PROGRAM Transformer
VAR_INPUT
	// reset signal for the error condition
	reset_error:		BOOL := FALSE;
	// signal to start the transformer
	softstart_trafo:	BOOL;
END_VAR
VAR_OUTPUT
	// indicates the phases for the hydraulics
	phase_available:	BOOL;
	// trafo failed to start after timeout
	power_failure:		BOOL;
	// restart was inhibited
	restart_inhibited:	BOOL;
END_VAR
VAR
	// watchdog for trafo softstarter
	power_watchdog: 	TON;
	// timer to measure the startup time
	power_timer:		FB_timer;
	// timeout for the startup
	startup_timeout:	TIME := T#5S;
	// error state
	power_error_state:	SR;
	// restart inhibitor
	restart_inhibit:	TOF;
	PowerEvent:			FB_EventLog;
	PowerLog:			FB_EventLog;
END_VAR

power_timer(bStart := GVL_Main.softstart_trafo, bStop := power_OK);
power_watchdog(IN := GVL_Main.softstart_trafo AND NOT power_OK,
				PT := startup_timeout,
				Q => power_failure);
power_error_state(SET1 := power_failure, RESET := reset_error);
restart_inhibit(IN := GVL_MAIN.trafo_bypassed, PT := T#5S);

restart_inhibited := NOT GVL_MAIN.trafo_bypassed AND restart_inhibit.Q;
IF restart_inhibited THEN
	softstart_trafo := FALSE;
END_IF
GVL_Main.softstart_trafo := softstart_trafo AND NOT error;

phase_available := TRUE; (*GVL_Main.L1L2_voltage > 360.0 AND
					GVL_Main.L2L3_voltage > 360.0 AND
					GVL_Main.L3L1_voltage > 360.0; *)

PowerEvent(	
	Trigger := 		power_failure, 
	Level := 		ADSLOG_MSGTYPE_ERROR,
	FormatString :=	'%s',
	OnMessage := 	'Servo power FAILURE!',
	OffMEssage := 	'Servo power OK');
PowerLog(	
	Trigger := 		power_OK, 
	Level := 		ADSLOG_MSGTYPE_HINT,
	FormatString :=	'%s',
	OnMessage := 	'Mains power is ON',
	OffMEssage := 	'Mains power is OFF');

PROPERTY error : BOOL
GET
error := power_error_state.Q1;
END_GET
END_PROPERTY

PROPERTY power_ok : BOOL
// indicates the power state for the AX5000
GET
power_ok := GVL_main.trafo_bypassed;
END_GET
END_PROPERTY

METHOD reset : BOOL
VAR_INPUT
END_VAR
IF error THEN
	reset_error := TRUE;
ELSE
	reset_error := FALSE;
END_IF
END_METHOD

METHOD start : BOOL
VAR_INPUT
END_VAR
softstart_trafo := TRUE;
END_METHOD

PROPERTY startup_time : TIME
GET
startup_time := power_timer.tDifference;
END_GET
SET
startup_timeout := startup_time;
END_SET
END_PROPERTY

METHOD stop : BOOL
VAR_INPUT
END_VAR
softstart_trafo := FALSE;
END_METHOD

END_PROGRAM

(* stored: Version 1.1.0.1, ProductVersion 3.1.4024.9
   POU Transformer: Id {0a280e03-5b4e-47d4-8865-661b3df896f8}, SpecialFunc None
   Property error: Id {4119c9eb-4956-4e1d-9bb0-76d34951f705}
   Get Get: Id {e45da732-7f2c-4a0e-907f-de39a5f0c547}
   Property power_ok: Id {b0563a1e-dd5f-461f-9fae-5a1c236a42b8}
   Get Get: Id {5f1a2942-c9ab-478b-ae9d-c8ca63749554}
   Method reset: Id {b8036108-f586-442e-9cc9-919ffec9b1dd}
   Method start: Id {a80781e7-508e-41b1-b8d1-4bd694cc587f}
   Property startup_time: Id {8d0359b7-73eb-49bc-a2c4-6389e6c8a8c3}
   Get Get: Id {9d98fddd-76c6-4d13-856d-d066f5e879ac}
   Set Set: Id {2a464548-0a55-47a9-a440-6ca3ebe43469}
   Method stop: Id {615c1e3c-bdce-41f6-a0af-3d3824c0fb9b} *)
